{attribute 'hide_all_locals'}
FUNCTION_BLOCK HaltMover EXTENDS TaskBase
VAR_INPUT
END_VAR
VAR_OUTPUT
END_VAR
VAR
	haltMover : Tc3_McCollisionAvoidance.MC_HaltCA;
	_axis : REFERENCE TO Tc2_MC2.AXIS_REF;
	_HaltMover : BOOL;
END_VAR

METHOD Abort : BOOL
haltMover.Execute := FALSE;
_busy := FALSE;
_HaltMover := FALSE;
Abort := TRUE;
State := 0;
END_METHOD

METHOD Cycle : BOOL
VAR_INPUT
END_VAR
CASE State OF
	0:
		IF _HaltMover THEN
			_done := FALSE;
			_error := FALSE;
			_busy := TRUE;
			haltMover.Execute := TRUE;
			IF haltMover.Busy THEN
				State := 10;
				_HaltMover := FALSE;
			END_IF
		END_IF
	
	10:
		IF NOT haltMover.Busy THEN
			IF haltMover.Done THEN
				_done := TRUE;
			ELSIF haltMover.Error THEN
				_error := TRUE;
			END_IF
			_busy := FALSE;
			haltMover.Execute := FALSE;
			State := 0;
		END_IF
END_CASE

haltMover(Axis := _axis);
END_METHOD

METHOD Execute : BOOL
VAR_INPUT
END_VAR
Execute := _HaltMover := true;
END_METHOD

METHOD FB_init : BOOL
VAR_INPUT
	bInitRetains : BOOL; // if TRUE, the retain variables are initialized (warm start / cold start)
	bInCopyCode : BOOL;  // if TRUE, the instance afterwards gets moved into the copy code (online change)
	axis : reference TO AXIS_REF;
END_VAR
_axis REF= axis;
END_METHOD

END_FUNCTION_BLOCK

(* stored: Version 1.1.0.1, ProductVersion 3.1.4024.12
   POU HaltMover: Id {16fe934f-2b92-45c5-becd-cbf7a242dbb1}, SpecialFunc None
   Method Abort: Id {48a4c415-0254-4332-8d1a-2734e5dda505}
   Method Cycle: Id {1e7367c4-25b5-40fa-b219-770d9b7044ce}
   Method Execute: Id {87eca2aa-365e-4c2f-b198-b62e8029fb82}
   Method FB_init: Id {0fd2927a-947b-415e-b53d-5482c2b0a045} *)
